// Mitsubishi GX Works2 project: ZP_funtion_EX2   PLC: Q03UDV

PROGRAM MAIN
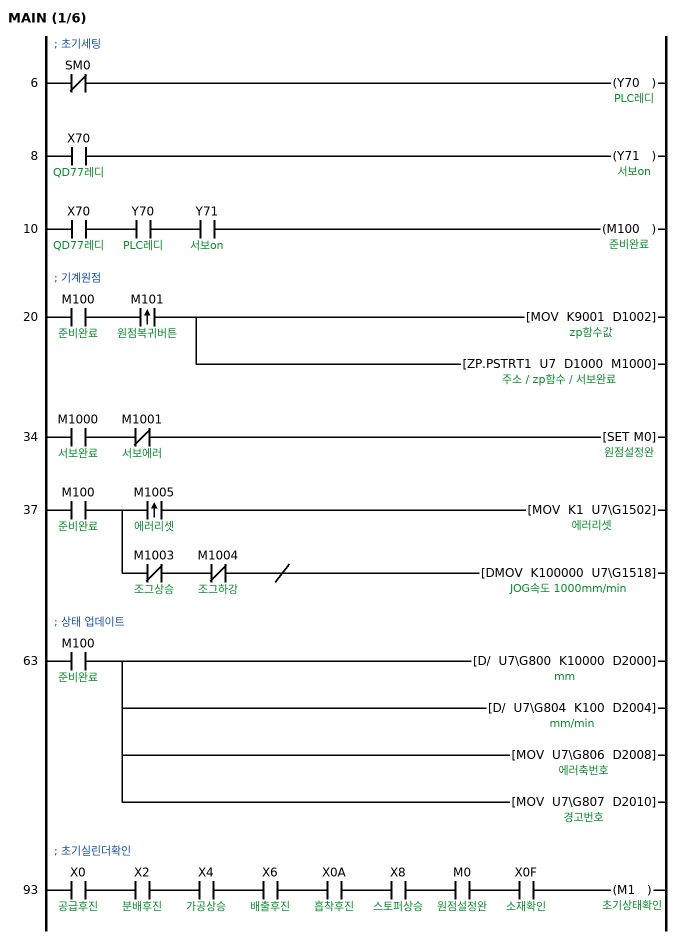
; 초기세팅
6     LDI     SM0
      OUT     Y70  ; PLC레디
8     LD      X70  ; QD77레디
      OUT     Y71  ; 서보on
10    LD      X70  ; QD77레디
      AND     Y70  ; PLC레디
      AND     Y71  ; 서보on
      OUT     M100  ; 준비완료
; 기계원점
20    LD      M100  ; 준비완료
      ANDP    M101  ; 원점복귀버튼
      MOV     K9001 D1002  ; zp함수값
      ZP.PSTRT1 U7 D1000 M1000  ; 주소 / zp함수 / 서보완료
34    LD      M1000  ; 서보완료
      ANI     M1001  ; 서보에러
      SET     M0  ; 원점설정완
37    LD      M100  ; 준비완료
      MPS
      ANDP    M1005  ; 에러리셋
      MOV     K1 U7\G1502  ; 에러리셋
      MPP
      ANI     M1003  ; 조그상승
      ANI     M1004  ; 조그하강
      INV
      DMOV    K100000 U7\G1518  ; JOG속도 1000mm/min
; 상태 업데이트
63    LD      M100  ; 준비완료
      D/      U7\G800 K10000 D2000  ; mm
      D/      U7\G804 K100 D2004  ; mm/min
      MOV     U7\G806 D2008  ; 에러축번호
      MOV     U7\G807 D2010  ; 경고번호
; 초기실린더확인
93    LD      X0  ; 공급후진
      AND     X2  ; 분배후진
      AND     X4  ; 가공상승
      AND     X6  ; 배출후진
      AND     X0A  ; 흡착후진
      AND     X8  ; 스토퍼상승
      AND     M0  ; 원점설정완
      AND     X0F  ; 소재확인
      OUT     M1  ; 초기상태확인
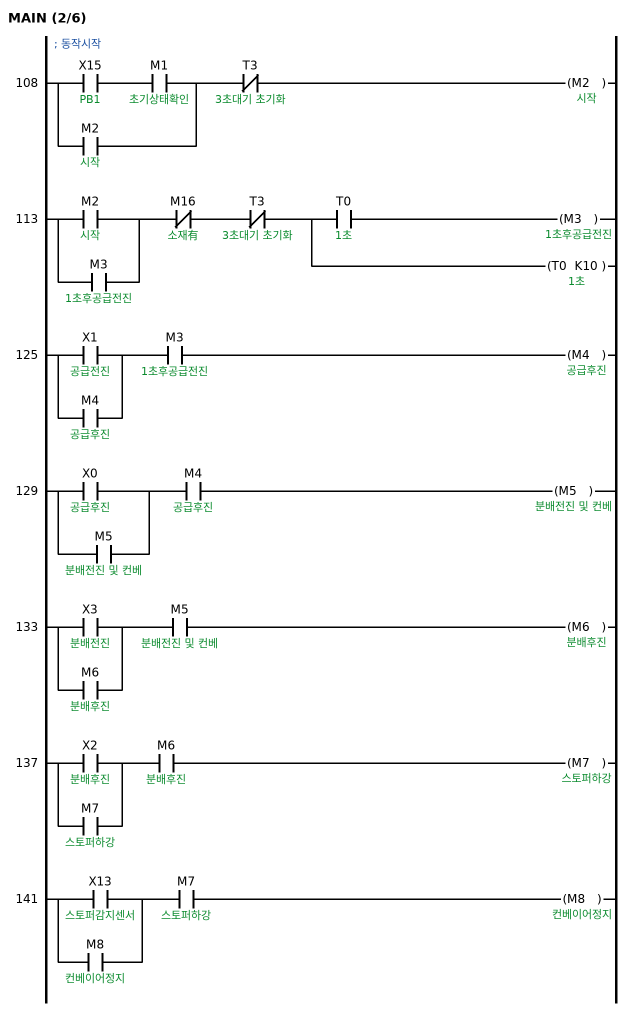
; 동작시작
108   LD      X15  ; PB1
      AND     M1  ; 초기상태확인
      OR      M2  ; 시작
      ANI     T3  ; 3초대기 초기화
      OUT     M2  ; 시작
113   LD      M2  ; 시작
      OR      M3  ; 1초후공급전진
      ANI     M16  ; 소재有
      ANI     T3  ; 3초대기 초기화
      MPS
      AND     T0  ; 1초
      OUT     M3  ; 1초후공급전진
      MPP
      OUT     T0 K10  ; 1초
125   LD      X1  ; 공급전진
      OR      M4  ; 공급후진
      AND     M3  ; 1초후공급전진
      OUT     M4  ; 공급후진
129   LD      X0  ; 공급후진
      OR      M5  ; 분배전진 및 컨베
      AND     M4  ; 공급후진
      OUT     M5  ; 분배전진 및 컨베
133   LD      X3  ; 분배전진
      OR      M6  ; 분배후진
      AND     M5  ; 분배전진 및 컨베
      OUT     M6  ; 분배후진
137   LD      X2  ; 분배후진
      OR      M7  ; 스토퍼하강
      AND     M6  ; 분배후진
      OUT     M7  ; 스토퍼하강
141   LD      X13  ; 스토퍼감지센서
      OR      M8  ; 컨베이어정지
      AND     M7  ; 스토퍼하강
      OUT     M8  ; 컨베이어정지
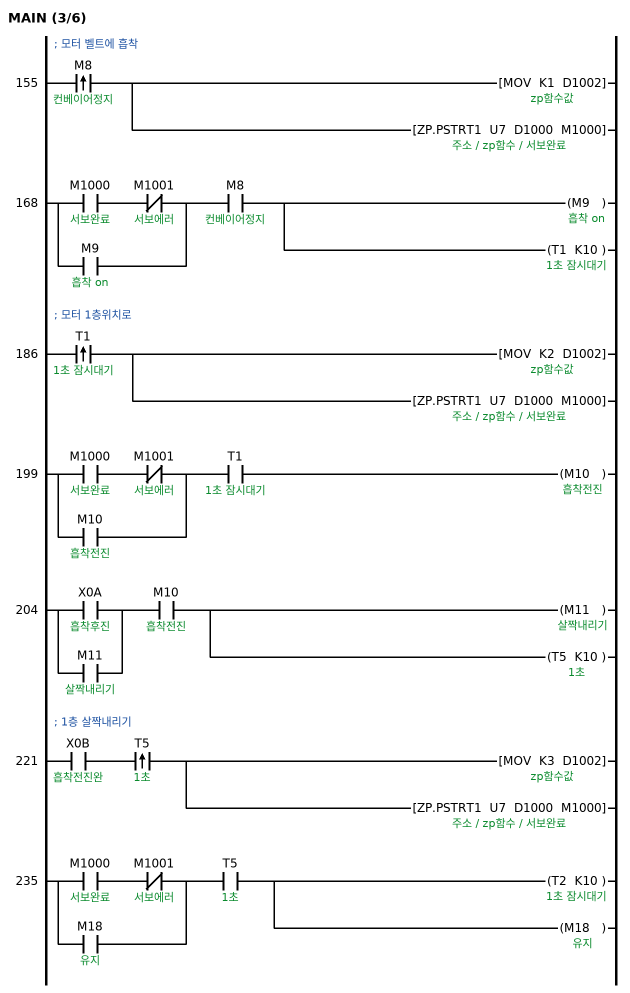
; 모터 벨트에 흡착
155   LDP     M8  ; 컨베이어정지
      MOV     K1 D1002
      ZP.PSTRT1 U7 D1000 M1000
168   LD      M1000  ; 서보완료
      ANI     M1001  ; 서보에러
      OR      M9  ; 흡착 on
      AND     M8  ; 컨베이어정지
      OUT     M9  ; 흡착 on
      OUT     T1 K10  ; 1초 잠시대기
; 모터 1층위치로
186   LDP     T1  ; 1초 잠시대기
      MOV     K2 D1002
      ZP.PSTRT1 U7 D1000 M1000
199   LD      M1000  ; 서보완료
      ANI     M1001  ; 서보에러
      OR      M10  ; 흡착전진
      AND     T1  ; 1초 잠시대기
      OUT     M10  ; 흡착전진
204   LD      X0A  ; 흡착후진
      OR      M11  ; 살짝내리기
      AND     M10  ; 흡착전진
      OUT     M11  ; 살짝내리기
      OUT     T5 K10  ; 1초
; 1층 살짝내리기
221   LD      X0B  ; 흡착전진완
      ANDP    T5  ; 1초
      MOV     K3 D1002
      ZP.PSTRT1 U7 D1000 M1000
235   LD      M1000  ; 서보완료
      ANI     M1001  ; 서보에러
      OR      M18  ; 유지
      AND     T5  ; 1초
      OUT     T2 K10  ; 1초 잠시대기
      OUT     M18  ; 유지
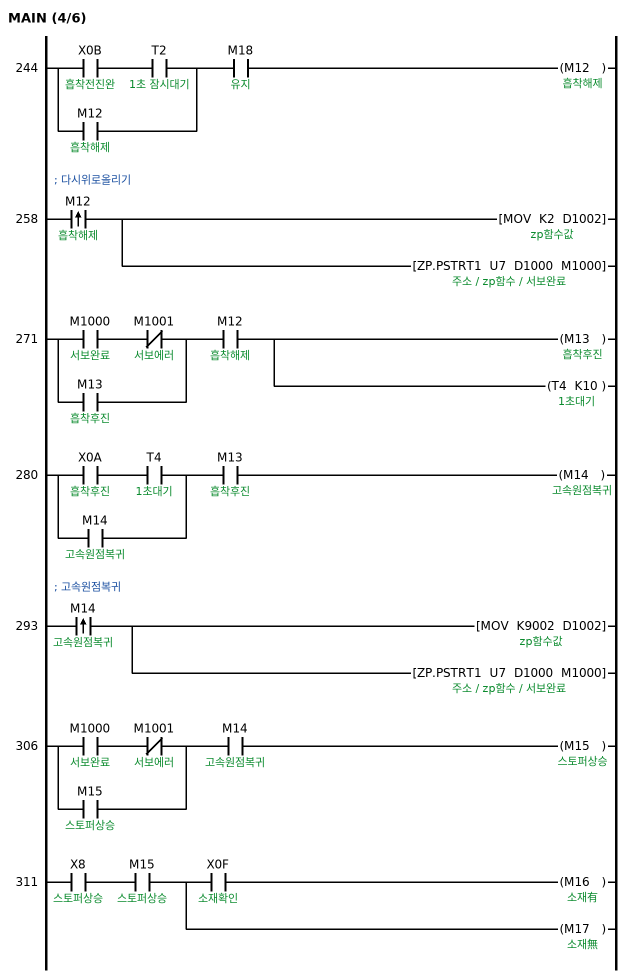
244   LD      X0B  ; 흡착전진완
      AND     T2  ; 1초 잠시대기
      OR      M12  ; 흡착해제
      AND     M18  ; 유지
      OUT     M12  ; 흡착해제
; 다시위로올리기
258   LDP     M12  ; 흡착해제
      MOV     K2 D1002
      ZP.PSTRT1 U7 D1000 M1000
271   LD      M1000  ; 서보완료
      ANI     M1001  ; 서보에러
      OR      M13  ; 흡착후진
      AND     M12  ; 흡착해제
      OUT     M13  ; 흡착후진
      OUT     T4 K10  ; 1초대기
280   LD      X0A  ; 흡착후진
      AND     T4  ; 1초대기
      OR      M14  ; 고속원점복귀
      AND     M13  ; 흡착후진
      OUT     M14  ; 고속원점복귀
; 고속원점복귀
293   LDP     M14  ; 고속원점복귀
      MOV     K9002 D1002
      ZP.PSTRT1 U7 D1000 M1000
306   LD      M1000  ; 서보완료
      ANI     M1001  ; 서보에러
      OR      M15  ; 스토퍼상승
      AND     M14  ; 고속원점복귀
      OUT     M15  ; 스토퍼상승
311   LD      X8  ; 스토퍼상승
      AND     M15  ; 스토퍼상승
      MPS
      AND     X0F  ; 소재확인
      OUT     M16  ; 소재有
      MPP
      OUT     M17  ; 소재無
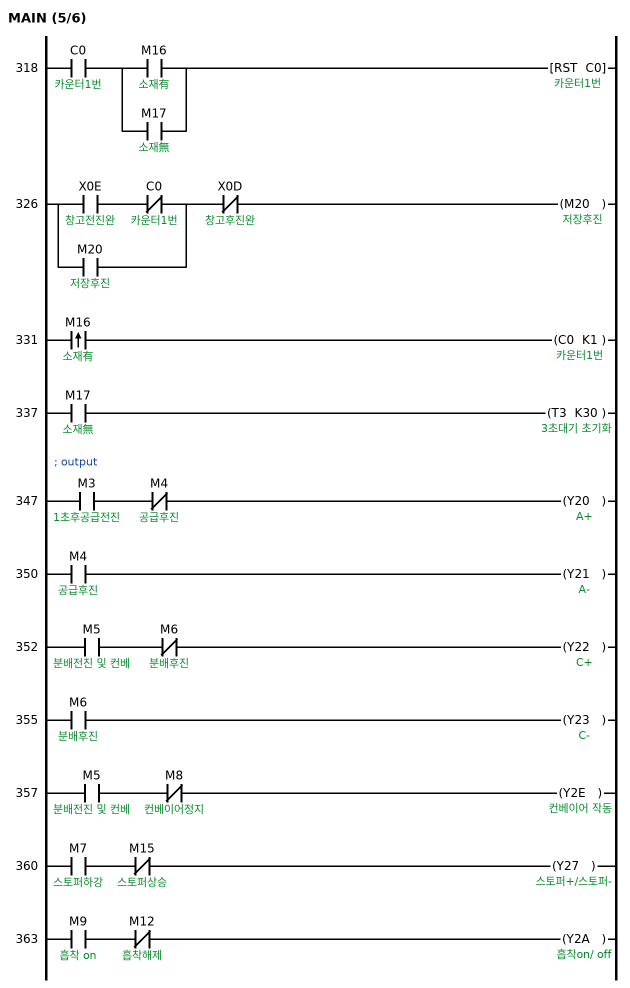
318   LD      C0  ; 카운터1번
      LD      M16  ; 소재有
      OR      M17  ; 소재無
      ANB
      RST     C0  ; 카운터1번
326   LD      X0E  ; 창고전진완
      ANI     C0  ; 카운터1번
      OR      M20  ; 저장후진
      ANI     X0D  ; 창고후진완
      OUT     M20  ; 저장후진
331   LDP     M16  ; 소재有
      OUT     C0 K1  ; 카운터1번
337   LD      M17  ; 소재無
      OUT     T3 K30  ; 3초대기 초기화
; output
347   LD      M3  ; 1초후공급전진
      ANI     M4  ; 공급후진
      OUT     Y20  ; A+
350   LD      M4  ; 공급후진
      OUT     Y21  ; A-
352   LD      M5  ; 분배전진 및 컨베
      ANI     M6  ; 분배후진
      OUT     Y22  ; C+
355   LD      M6  ; 분배후진
      OUT     Y23  ; C-
357   LD      M5  ; 분배전진 및 컨베
      ANI     M8  ; 컨베이어정지
      OUT     Y2E  ; 컨베이어 작동
360   LD      M7  ; 스토퍼하강
      ANI     M15  ; 스토퍼상승
      OUT     Y27  ; 스토퍼+/스토퍼-
363   LD      M9  ; 흡착 on
      ANI     M12  ; 흡착해제
      OUT     Y2A  ; 흡착on/ off
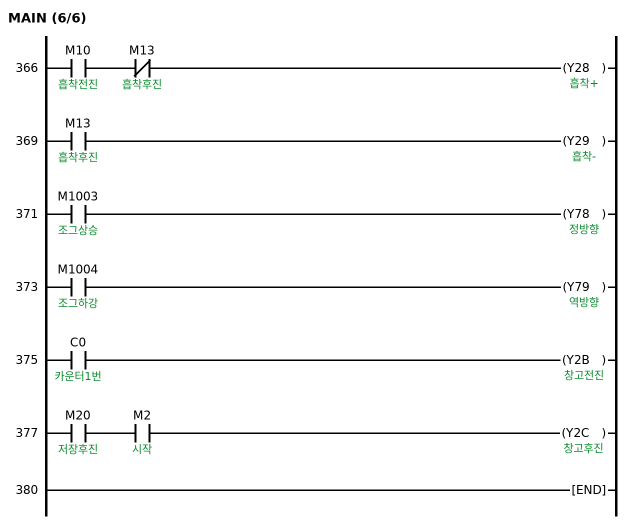
366   LD      M10  ; 흡착전진
      ANI     M13  ; 흡착후진
      OUT     Y28  ; 흡착+
369   LD      M13  ; 흡착후진
      OUT     Y29  ; 흡착-
371   LD      M1003  ; 조그상승
      OUT     Y78  ; 정방향
373   LD      M1004  ; 조그하강
      OUT     Y79  ; 역방향
375   LD      C0  ; 카운터1번
      OUT     Y2B  ; 창고전진
377   LD      M20  ; 저장후진
      AND     M2  ; 시작
      OUT     Y2C  ; 창고후진
380   END
END_PROGRAM

// device comments not shown above
X9  ; 스토퍼하강
M19  ; 두번째 재료 전진
